// TIA Portal V19 export
DATA_BLOCK "PPrgArchive5"   // DB509
// stored: IsOnlyStoredInLoadMemory true, MemoryReserve 0, Namespace G
   VAR RETAIN
      PRG : Array[401..500] of "PPrg_Data";
   END_VAR
BEGIN
END_DATA_BLOCK
